FUNCTION_BLOCK FB_BrakesRearm
VAR_INPUT
END_VAR
VAR_OUTPUT
END_VAR
VAR
END_VAR

END_FUNCTION_BLOCK

(* stored: Version 1.1.0.1
   POU FB_BrakesRearm: Id {1a49c53a-438a-46aa-b7dc-e596bb02d16b}, SpecialFunc None *)
